FUNCTION F_TaskTime : LREAL
VAR
	TaskIndex: DINT;
END_VAR

TaskIndex := GETCURTASKINDEXEX();
IF TaskIndex > 0 THEN
    F_TaskTime := UDINT_TO_LREAL(TwinCAT_SystemInfoVarList._taskInfo[TaskIndex].CycleTime) * LREAL#1E-7;
END_IF

END_FUNCTION

(* stored: Version 1.1.0.1, ProductVersion 3.1.4024.9
   POU F_TaskTime: Id {834bffb3-5daf-44ca-aaaf-12e71bd9f640}, SpecialFunc None *)
